{attribute 'qualified_only'}
{attribute 'strict'}
TYPE E_Huawei_SmartLogger_Error :
(
	eNoError := 0,
	eModbusTCPError := 1,
	eHuawei_SmartLoggerError := 2,
	eHuawei_SmartLoggerTooBigValueReceived := 3
);
END_TYPE

(* stored: Version 1.1.0.1, ProductVersion 3.1.4024.11
   DUT E_Huawei_SmartLogger_Error: Id {eb6e91ed-ef17-4119-b65b-862acd9b418e} *)
